      4:
        _nAx                          := _nAx + 1;
        _eState                       := E_PROGRESS.PROGRESS_BUSY;
        _fbGearInMultiMaster.Master4  := _Axes[_nMasterIndex[4]];   // assign AXIS_REF of master
    ELSE
      _eState                         := E_PROGRESS.PROGRESS_CHECK;
    END_CASE
END_CASE
CASE _eState
OF
  E_PROGRESS.PROGRESS_CHECK:
    _fbGearInMultiMaster(
                      Slave           := _AxisRef, 
                      Enable          := TRUE, 
                      GearRatio1      := _GearInParameter^[_nAxisIndex].rGearRatio[1], 
                      GearRatio2      := _GearInParameter^[_nAxisIndex].rGearRatio[2], 
                      GearRatio3      := _GearInParameter^[_nAxisIndex].rGearRatio[3], 
                      GearRatio4      := _GearInParameter^[_nAxisIndex].rGearRatio[4], 
                      Acceleration    := _GearInParameter^[_nAxisIndex].Acceleration, 
                      Deceleration    := _GearInParameter^[_nAxisIndex].Deceleration, 
                      Jerk            := _GearInParameter^[_nAxisIndex].Jerk);

    IF (_fbGearInMultiMaster.Error)
    THEN
      _nErr                           := _fbGearInMultiMaster.ErrorID;
      _stMsg.eType                    := E_MessageType.eMessageError;
      _stMsg.eDevice                  := e_Device.Axis + TO_UINT(_AxisRef.NcToPlc.AxisId);
      _stMsg.eSubdevice               := e_Subdevice.fbGearInMultiMaster;
      _stMsg.iErrorNumber             := _nErr;

      _stMsg.sText                    := concat(TO_STRING(_eCmd),'[');
      _stMsg.sText                    := concat(_stMsg.sText, TO_STRING(_nAxisIndex));
      _stMsg.sText                    := concat(_stMsg.sText, ']');
      _stMsg.sText                    := concat('fbGearInMultiMaster error: ', TO_STRING(_nErr));
      f_MessageSet(_stMsg);
      _eState                         := E_PROGRESS.PROGRESS_ERROR;

    ELSIF (_fbGearIn.InGear)
    THEN
      _eState                         := E_PROGRESS.PROGRESS_WORKING;
    END_IF

END_CASE
CASE _eState
OF
  E_PROGRESS.PROGRESS_WORKING:
    // now GearRatio[x] can be altered from outside
    // axis function waits here for further instructions from outside world
    // _stCtrl[_nAxisIndex].eProgress = e_Progress.DONE must be used to leave this axis function
    _fbGearInMultiMaster(
                      Slave           := _AxisRef, 
                      Enable          := TRUE, 
                      GearRatio1      := _GearInParameter^[_nAxisIndex].rGearRatio[1], 
                      GearRatio2      := _GearInParameter^[_nAxisIndex].rGearRatio[2], 
                      GearRatio3      := _GearInParameter^[_nAxisIndex].rGearRatio[3], 
                      GearRatio4      := _GearInParameter^[_nAxisIndex].rGearRatio[4], 
                      Acceleration    := _GearInParameter^[_nAxisIndex].Acceleration, 
                      Deceleration    := _GearInParameter^[_nAxisIndex].Deceleration, 
                      Jerk            := _GearInParameter^[_nAxisIndex].Jerk);

    IF (_fbGearInMultiMaster.Error)
    THEN
      _nErr                           := _fbGearInMultiMaster.ErrorID;
      _stMsg.eType                    := E_MessageType.eMessageError;
      _stMsg.eDevice                  := e_Device.Axis + TO_UINT(_AxisRef.NcToPlc.AxisId);
      _stMsg.eSubdevice               := e_Subdevice.fbGearInMultiMaster;
      _stMsg.iErrorNumber             := _nErr;

      _stMsg.sText                    := concat(TO_STRING(_eCmd),'[');
      _stMsg.sText                    := concat(_stMsg.sText, TO_STRING(_nAxisIndex));
      _stMsg.sText                    := concat(_stMsg.sText, ']');
      _stMsg.sText                    := concat('fbGearInMultiMaster error: ', TO_STRING(_nErr));
      f_MessageSet(_stMsg);
      _eState                         := E_PROGRESS.PROGRESS_ERROR;

    ELSIF (_Ctrl^[_nAxisIndex].eProgress = E_PROGRESS.PROGRESS_DONE)
    THEN
      // when Ctrl decides to leave; make finishing move and be done
      _eState                         := E_PROGRESS.PROGRESS_STILL_WORKING;
    END_IF
END_CASE
CASE _eState
OF
  E_PROGRESS.PROGRESS_STILL_WORKING:
    _eState                           := E_PROGRESS.PROGRESS_DONE;

    _stMsg.eType                      := E_MessageType.eMessageInfo;
    _stMsg.eDevice                    := e_Device.Axis + TO_UINT(_AxisRef.NcToPlc.AxisId);
    _stMsg.eSubdevice                 := e_Subdevice.fbGearInMultiMaster;
    _stMsg.iErrorNumber               := _eState;

    _stMsg.sText                      := concat(TO_STRING(_eCmd), ': ');
    _stMsg.sText                      := concat(_stMsg.sText, TO_STRING(_eState));
    f_MessageSet(_stMsg);
END_CASE

AxisGearInMultiMaster                 := _eState;
END_METHOD

PROPERTY AxisGearInParameter : pointer to ARRAY[1..PLC_CONSTANT.MAX_AXIS] OF ST_GEAR_IN
SET
_GearInParameter := AxisGearInParameter;
END_SET
END_PROPERTY

METHOD AxisGearOut : E_PROGRESS
VAR_INPUT
  Execute           : BOOL;
END_VAR
VAR_INST
  _eState           : E_PROGRESS;
  _rValue           : LREAL;
  _nErr             : UDINT;
  _stMsg            : ST_Message;
END_VAR
IF NOT Check() THEN AxisGearOut := E_PROGRESS.PROGRESS_ERROR; RETURN; END_IF
IF NOT Execute THEN _eState := E_PROGRESS.PROGRESS_INIT; END_IF

CASE _eState
OF
  E_PROGRESS.PROGRESS_INIT:
    IF Execute 
    THEN
      memset(ADR(_stMsg),0,SIZEOF(_stMsg));
      _nErr                       := 0;
      _rValue                     := 0;

      _fbGearOut(
            Slave                 := _AxisRef, 
            Execute               := FALSE);

      IF (_AxisRef.NcToPlc.CoupleState < 2)
      THEN
        _eState                   := E_PROGRESS.PROGRESS_DONE;
      ELSE
        _eState                   := E_PROGRESS.PROGRESS_BUSY;

        _stMsg.eType              := E_MessageType.eMessageInfo;
        _stMsg.eDevice            := e_Device.Axis + TO_UINT(_AxisRef.NcToPlc.AxisId);
        _stMsg.eSubdevice         := e_Subdevice.fbGearOut;
        _stMsg.iErrorNumber       := 0;
  
        _stMsg.sText              := concat('GearOut BUSY: ', TO_STRING(_nAxisIndex));
        f_MessageSet(_stMsg);
      END_IF
    END_IF
END_CASE
CASE _eState
OF
  E_PROGRESS.PROGRESS_BUSY:
    _fbGearOut(
            Slave                 := _AxisRef, 
            Execute               := TRUE);

    IF (_fbGearOut.Error)
    THEN
      _nErr                       := _fbGearOut.ErrorID;

      _stMsg.eType                := E_MessageType.eMessageError;
      _stMsg.eDevice              := e_Device.Axis + TO_UINT(_AxisRef.NcToPlc.AxisId);
      _stMsg.eSubdevice           := e_Subdevice.fbGearOut;
      _stMsg.iErrorNumber         := _nErr;

      _stMsg.sText                := concat('GearOut ERROR: ', TO_STRING(_nAxisIndex));
      f_MessageSet(_stMsg);
      _eState                     := E_PROGRESS.PROGRESS_ERROR;

    ELSIF (_fbGearOut.Done)
    THEN
      _stMsg.eType                := E_MessageType.eMessageInfo;
      _stMsg.eDevice              := e_Device.Axis + TO_UINT(_AxisRef.NcToPlc.AxisId);
      _stMsg.eSubdevice           := e_Subdevice.fbGearOut;
      _stMsg.iErrorNumber         := 0;
  
      _stMsg.sText                := concat('GearOut DONE: ', TO_STRING(_nAxisIndex));
      f_MessageSet(_stMsg);

      IF (_AxisRef.NcToPlc.CoupleState < 2)
      THEN
        _eState                   := E_PROGRESS.PROGRESS_DONE;
      ELSE
        _eState                   := E_PROGRESS.PROGRESS_STARTUP;
      END_IF
    END_IF
END_CASE
CASE _eState
OF
  E_PROGRESS.PROGRESS_STARTUP:
    _eState                       := E_PROGRESS.PROGRESS_BUSY;
    _fbGearOut(
          Slave                   := _AxisRef, 
          Execute                 := FALSE);

    _stMsg.eType                  := E_MessageType.eMessageInfo;
    _stMsg.eDevice                := e_Device.Axis + TO_UINT(_AxisRef.NcToPlc.AxisId);
    _stMsg.eSubdevice             := e_Subdevice.fbGearOut;
    _stMsg.iErrorNumber           := 0;

    _stMsg.sText                  := concat('GearOut CoupleState: ', TO_STRING(_AxisRef.NcToPlc.CoupleState));
    f_MessageSet(_stMsg);
END_CASE
CASE _eState
OF
  E_PROGRESS.PROGRESS_DONE,
  E_PROGRESS.PROGRESS_ERROR:
    _fbGearOut(
            Slave                 := _AxisRef, 
            Execute               := FALSE);
END_CASE

AxisGearOut                       := _eState;
END_METHOD

METHOD AxisHalt : E_PROGRESS
VAR_INPUT
  Execute           : BOOL;
  Data              : ST_AXIS_MOVE_DATA;
END_VAR
VAR_INST
  _eres,
  _eState           : E_PROGRESS;
  _rValue           : LREAL;
  _udiErr           : UDINT;
  _stMsg            : ST_Message;


END_VAR
IF NOT Check() THEN AxisHalt := E_PROGRESS.PROGRESS_ERROR; RETURN; END_IF
IF NOT Execute THEN _eState := E_PROGRESS.PROGRESS_INIT; END_IF

CASE _eState
OF
  E_PROGRESS.PROGRESS_INIT:
    IF Execute 
    THEN
      memset(ADR(_stMsg),0,SIZEOF(_stMsg));
      _udiErr       := 0;
      _rValue       := 0;
      _eState       := E_PROGRESS.PROGRESS_BUSY;
    END_IF
END_CASE
CASE _eState
OF
  E_PROGRESS.PROGRESS_BUSY:
    _eState         := E_PROGRESS.PROGRESS_OCCUPIED;
    _eres           := Halt(
                            Execute := FALSE, 
                            Dec     := Data.rDec, 
                            Jerk    := Data.rJerk);
END_CASE
CASE _eState
OF
  E_PROGRESS.PROGRESS_OCCUPIED:
    _eres           := Halt(
                            Execute := TRUE, 
                            Dec     := Data.rDec, 
                            Jerk    := Data.rJerk);

    IF (_eres = E_PROGRESS.PROGRESS_ERROR)
    THEN
        _eState     := E_PROGRESS.PROGRESS_ERROR;
    ELSIF (_eres = E_PROGRESS.PROGRESS_DONE)
    THEN 
      _eState       := E_PROGRESS.PROGRESS_WORKING;
    END_IF
END_CASE
CASE _eState
OF
  E_PROGRESS.PROGRESS_WORKING:
    _eState         := E_PROGRESS.PROGRESS_DONE;
    _eres           := Halt(
                            Execute := FALSE, 
                            Dec     := Data.rDec, 
                            Jerk    := Data.rJerk);
END_CASE

AxisHalt := _eState;
END_METHOD

METHOD AxisHome : E_PROGRESS
VAR_INPUT
  Execute           : BOOL;
END_VAR
VAR_INST
  _eres,
  _eState           : E_PROGRESS;
  _rValue           : LREAL;
  _udiErr           : UDINT;
  _stMsg            : ST_Message;


END_VAR
IF NOT Check() THEN AxisHome := E_PROGRESS.PROGRESS_ERROR; RETURN; END_IF
IF NOT Execute THEN _eState := E_PROGRESS.PROGRESS_INIT; END_IF

CASE _eState
OF
  E_PROGRESS.PROGRESS_INIT:
    IF Execute 
    THEN
      memset(ADR(_stMsg),0,SIZEOF(_stMsg));
      _udiErr               := 0;
      _rValue               := 0;

      IF (_AxisRef.Status.Homed)
      THEN
        _eState             := E_PROGRESS.PROGRESS_BUSY;
      ELSE
        _eState             := E_PROGRESS.PROGRESS_PREPARE;
      END_IF
    END_IF
END_CASE
CASE _eState
OF
  E_PROGRESS.PROGRESS_BUSY:
    _eState                 := E_PROGRESS.PROGRESS_STARTUP;
    _eres                   := Home(
                                    Execute   := FALSE,
                                    Position  := _HomeParameter^[_nAxisIndex].stHomingParam.Position,
                                    HomingMode:= Tc2_MC2.MC_HomingMode.MC_ResetCalibration,
                                    Options   := _HomeParameter^[_nAxisIndex].stHomingParam.Options);
END_CASE
CASE _eState
OF
  E_PROGRESS.PROGRESS_STARTUP:
    _Info^[_nAxisIndex].bReferenced   := FALSE;

    _eres                   := Home(
                                    Execute   := TRUE,
                                    Position  := _HomeParameter^[_nAxisIndex].stHomingParam.Position,
                                    HomingMode:= Tc2_MC2.MC_HomingMode.MC_ResetCalibration,
                                    Options   := _HomeParameter^[_nAxisIndex].stHomingParam.Options);
    IF (_eres = E_PROGRESS.PROGRESS_DONE)
    THEN
      _eState               := E_PROGRESS.PROGRESS_PREPARE;
    END_IF
END_CASE
CASE _eState
OF
  E_PROGRESS.PROGRESS_PREPARE:
      _eState               := E_PROGRESS.PROGRESS_CHECK;

      _eres                 := Home(
                                    Execute   := FALSE,
                                    Position  := _HomeParameter^[_nAxisIndex].stHomingParam.Position,
                                    HomingMode:= Tc2_MC2.MC_HomingMode.MC_ResetCalibration,
                                    Options   := _HomeParameter^[_nAxisIndex].stHomingParam.Options);
END_CASE
CASE _eState
OF
  E_PROGRESS.PROGRESS_CHECK:
    _eState                 := E_PROGRESS.PROGRESS_OCCUPIED;

END_CASE
CASE _eState
OF
  E_PROGRESS.PROGRESS_OCCUPIED:
    _eres                   := Home(
                                    Execute   := TRUE,
                                    Position  := _HomeParameter^[_nAxisIndex].stHomingParam.Position,
                                    HomingMode:= _HomeParameter^[_nAxisIndex].stHomingParam.HomingMode,
                                    Options   := _HomeParameter^[_nAxisIndex].stHomingParam.Options);

    IF (_eres = E_PROGRESS.PROGRESS_ERROR)
    THEN
      _eState               := E_PROGRESS.PROGRESS_ERROR;
    ELSIF (_eres = E_PROGRESS.PROGRESS_DONE)
    THEN
      _eState               := E_PROGRESS.PROGRESS_WORKING;
    END_IF
END_CASE
CASE _eState
OF
  E_PROGRESS.PROGRESS_WORKING:
    _eState                 := E_PROGRESS.PROGRESS_DONE;

    _eres                   := Home(
                                    Execute   := FALSE,
                                    Position  := _HomeParameter^[_nAxisIndex].stHomingParam.Position,
                                    HomingMode:= _HomeParameter^[_nAxisIndex].stHomingParam.HomingMode,
                                    Options   := _HomeParameter^[_nAxisIndex].stHomingParam.Options);
END_CASE

AxisHome := _eState;
END_METHOD

METHOD AxisIdle : E_PROGRESS
VAR_INPUT
  Execute           : BOOL;
END_VAR
VAR_INST
  _eResult,
  _eState           : E_PROGRESS;
  _stMsg            : ST_Message;
  _nRetry           : UINT;
END_VAR
IF NOT Check() THEN AxisIdle := E_PROGRESS.PROGRESS_ERROR; return; END_IF
IF NOT Execute THEN _eState := E_PROGRESS.PROGRESS_INIT; END_IF

CASE _eState
OF
  E_PROGRESS.PROGRESS_INIT:
    IF Execute 
    THEN
      memset(ADR(_stMsg),0,SIZEOF(_stMsg));
      _nRetry                       := 0;
      _eResult                      := Reset(FALSE);
      _eState                       := E_PROGRESS.PROGRESS_BUSY;
    END_IF
END_CASE
CASE _eState
OF
  E_PROGRESS.PROGRESS_BUSY:
    _eResult                        := Reset(TRUE);

    IF (_eResult = E_PROGRESS.PROGRESS_DONE)
    THEN
      _nRetry                       := _nRetry + 1;
      _eState                       := E_PROGRESS.PROGRESS_STARTUP;
    END_IF
END_CASE
CASE _eState
OF
  E_PROGRESS.PROGRESS_STARTUP:
    _eResult                        := Reset(FALSE);
    _eResult                        := Enable(FALSE);
    _eState                         := E_PROGRESS.PROGRESS_CHECK;
END_CASE
CASE _eState
OF
  E_PROGRESS.PROGRESS_PREPARE:
    _eResult                        := Reset(FALSE);
    _eResult                        := Enable(FALSE);

    _eState                         := E_PROGRESS.PROGRESS_BUSY;

    _stMsg.eType                    := E_MessageType.eMessageInfo;
    _stMsg.eDevice                  := e_Device.Axis + (_AxisRef.NcToPlc.AxisId);
    _stMsg.eSubdevice               :=  e_SubDevice.AxisIdle;
    _stMsg.iErrorNumber             := _nErrorId;

    _stMsg.sText                    := concat(TO_STRING(_eCmd), ' retry: ');
    _stMsg.sText                    := concat(_stMsg.sText, TO_STRING(_nRetry));

    f_MessageSet(_stMsg);
END_CASE
CASE _eState
OF
  E_PROGRESS.PROGRESS_CHECK:
    _eResult                        := Enable(TRUE);

    IF (_nRetry > MAX_RETRY)
    THEN
      _eState                       := E_PROGRESS.PROGRESS_ERROR;

    ELSIF (_eResult = E_PROGRESS.PROGRESS_DONE)
    THEN
      Enable(FALSE);
      _eState                       := E_PROGRESS.PROGRESS_DONE;

    ELSIF (_eResult = E_PROGRESS.PROGRESS_ERROR)
    THEN
      _eState                       := E_PROGRESS.PROGRESS_PREPARE;

      _nErrorId                     := _AxisRef.NcToPlc.ErrorCode;
    
      _stMsg.eType                  := E_MessageType.eMessageError;
      _stMsg.eDevice                := e_Device.Axis + (_AxisRef.NcToPlc.AxisId);
      _stMsg.eSubdevice             :=  e_SubDevice.AxisIdle;
      _stMsg.iErrorNumber           := _nErrorId;

      _stMsg.sText                  := concat(TO_STRING(_eCmd), ' error axis enable: ');
      _stMsg.sText                  := concat(_stMsg.sText, TO_STRING(_nAxisIndex));

      f_MessageSet(_stMsg);
    END_IF
END_CASE

AxisIdle                                := _eState;
END_METHOD

PROPERTY AxisIndex : uint
SET
_nAxisIndex := AxisIndex;
END_SET
END_PROPERTY

PROPERTY AxisInfo : pointer to ARRAY[1..PLC_CONSTANT.MAX_AXIS] OF ST_AXIS_INFO
SET
_Info := AxisInfo;
END_SET
END_PROPERTY

METHOD PRIVATE AxisInit : E_PROGRESS
VAR_INPUT
  Execute           : BOOL;
END_VAR
VAR_INST
  _eResult,
  _eState           : E_PROGRESS;
  _rValue           : LREAL;
  _stMsg            : ST_Message;
END_VAR
IF NOT Check() THEN AxisInit := E_PROGRESS.PROGRESS_ERROR; RETURN; END_IF
IF NOT Execute THEN _eState := E_PROGRESS.PROGRESS_INIT; END_IF

CASE _eState
OF
  E_PROGRESS.PROGRESS_INIT:
    IF Execute 
    THEN
      memset(ADR(_stMsg),0,SIZEOF(_stMsg));

      _nErrorId                     := 0;
      _rValue                       := 0;
      _eState                       := E_PROGRESS.PROGRESS_BUSY;
      _eInit                        := _eState;
    END_IF
END_CASE
CASE _eState
OF
  E_PROGRESS.PROGRESS_BUSY:
    _eState                         := E_PROGRESS.PROGRESS_STARTUP;
    _eResult                        := StartUp(FALSE);
END_CASE
CASE _eState
OF
  E_PROGRESS.PROGRESS_STARTUP:
    _eResult                        := StartUp(TRUE);
    IF (_eResult = E_PROGRESS.PROGRESS_DONE)
    THEN
      _eState                       := E_PROGRESS.PROGRESS_PREPARE;
      _eResult                      := AxisReset(FALSE);
    ELSIF (_eResult = E_PROGRESS.PROGRESS_ERROR)
    THEN
      _eState                       := _eResult;

      _stMsg.eType                  := E_MessageType.eMessageError;
      _stMsg.eDevice                := e_Device.Axis + (_AxisRef.NcToPlc.AxisId);
      _stMsg.eSubdevice             := e_Subdevice.AxisStartUp;
      _stMsg.iErrorNumber := _nErrorId  := 6666;

      _stMsg.sText                  := TO_STRING(_eState);
      f_MessageSet(_stMsg);

    END_IF
END_CASE
CASE _eState
OF
  E_PROGRESS.PROGRESS_PREPARE:
    _eResult                        := AxisReset(TRUE);
    IF (_eResult = E_PROGRESS.PROGRESS_DONE)
    THEN
      _fbCoeRead(
                Execute             := FALSE,
                NetId               := _AxisRef.ADS.NetId, 
                Axis                := _AxisRef);
  
      IF (EncoderType > 1)
      THEN
        memset(ADR(_sDeviceName),0,SIZEOF(_sDeviceName));
  
        _eState                     := E_PROGRESS.PROGRESS_CHECK;
      ELSE
        _sDeviceName                := _sAxisName;
        _eState                     := E_PROGRESS.PROGRESS_WORKING;
      END_IF
    ELSIF (_eResult = E_PROGRESS.PROGRESS_ERROR)
    THEN
      _eState                       := _eResult;

      _stMsg.eType                  := E_MessageType.eMessageError;
      _stMsg.eDevice                := e_Device.Axis + (_AxisRef.NcToPlc.AxisId);
      _stMsg.eSubdevice             := e_Subdevice.AxisStartUp;
      _stMsg.iErrorNumber           := ErrorId;

      _stMsg.sText                  := TO_STRING(_eState);
      f_MessageSet(_stMsg);

    END_IF
END_CASE
CASE _eState
OF
  E_PROGRESS.PROGRESS_CHECK:
    _eResult                        := AxisReset(FALSE);
    // get manufacturer device name in CoE
    _fbCoeRead.Index                := 16#1008;
    _fbCoeRead.SubIndex             := 0;
    _fbCoeRead.pDstBuf              := ADR(_sDeviceName);
    _fbCoeRead.BufLen               := SIZEOF(_sDeviceName);

    _fbCoeRead(
              Execute               := TRUE,
              NetId                 := _AxisRef.ADS.NetId, 
              Axis                  := _AxisRef);

    IF _fbCoeRead.Busy
    THEN
      _eState                       := E_PROGRESS.PROGRESS_OCCUPIED;
    END_IF
END_CASE
CASE _eState
OF
  E_PROGRESS.PROGRESS_OCCUPIED:
    _fbCoeRead(
              NetId                 := _AxisRef.ADS.NetId, 
              Axis                  := _AxisRef);

    IF NOT _fbCoeRead.Busy
    THEN
      _eState                       := E_PROGRESS.PROGRESS_WORKING;
    END_IF

// in case encoder type is used without hardware, error must be ignored here
(*
    IF (_fbCoeRead.Error)
    THEN
      _eState                       := E_PROGRESS.ERROR;

      _Info^[_nAxisIndex].nErrorId  := SEL((_fbCoeRead.CANopenErrId > 0), _fbCoeRead.AdsErrId, _fbCoeRead.CANopenErrId);

      _stMsg.eType                  := E_MessageType.eMessageError;
      _stMsg.eDevice                := e_Device.Axis + TO_DINT(_AxisRef.NcToPlc.AxisId);
      _stMsg.eSubdevice             := e_Subdevice.fbCoeRead;

      _stMsg.iErrorNumber           := SEL((_fbCoeRead.CANopenErrId > 0), _fbCoeRead.AdsErrId, _fbCoeRead.CANopenErrId);

      _stMsg.sText                  := TO_STRING(_eState);
      f_MessageSet(_stMsg);

      _fbCoeRead(
                Execute             := FALSE,
                NetId               := _AxisRef.ADS.NetId, 
                Axis                := _AxisRef);

    ELSIF NOT _fbCoeRead.Busy
    THEN
      _eState                       := E_PROGRESS.WORKING;
    END_IF
*)
END_CASE
CASE _eState
OF
  E_PROGRESS.PROGRESS_WORKING:
    _eState                         := E_PROGRESS.PROGRESS_DONE;
    // set default for axis release
    AxisEnableNegative              := TRUE;
    AxisEnablePositive              := TRUE;

    // clear fb
    _fbCoeRead(
              Execute               := FALSE,
              NetId                 := _AxisRef.ADS.NetId, 
              Axis                  := _AxisRef);

    _stMsg.eType                    := E_MessageType.eMessageInfo;
    _stMsg.eDevice                  := e_Device.Axis + (_AxisRef.NcToPlc.AxisId);
    _stMsg.eSubdevice               := e_Subdevice.AxisStartUp;
    _stMsg.iErrorNumber             := 0;
    _stMsg.sText                    := concat('Axis Init: ', _sDeviceName);
    _stMsg.sText                    := concat(_stMsg.sText, ' : ');
    _stMsg.sText                    := concat(_stMsg.sText, TO_STRING(_eState));

  IF (_MessageLevel > E_MessageType.eMessageError)
  THEN
    f_MessageSet(_stMsg);
  END_IF
END_CASE

AxisInit                            := _eState;
END_METHOD

METHOD AxisMoveToPosition : E_PROGRESS
VAR_INPUT
  Execute           : BOOL;
  Data              : ST_AXIS_MOVE_DATA;
END_VAR
VAR_INST
  _eres,
  _eState           : E_PROGRESS;
END_VAR
IF NOT Check() THEN AxisMoveToPosition := E_PROGRESS.PROGRESS_ERROR; RETURN; END_IF
IF NOT Execute THEN _eState := E_PROGRESS.PROGRESS_INIT; END_IF

CASE _eState
OF
  E_PROGRESS.PROGRESS_INIT:
    IF Execute 
    THEN
      _eState               := E_PROGRESS.PROGRESS_BUSY;
    END_IF
END_CASE
CASE _eState
OF
  E_PROGRESS.PROGRESS_BUSY:
    _eState                 := E_PROGRESS.PROGRESS_OCCUPIED;
    _eres                   := MoveToPos(
                                      Execute    := FALSE, 
                                      Position   := Data.rSetPos, 
                                      Vel        := Data.rSetVelo, 
                                      Acc        := Data.rAcc, 
                                      Dec        := Data.rDec, 
                                      Jerk       := Data.rJerk, 
                                      BufferMode := Tc2_MC2.MC_BufferMode.MC_Aborting);
END_CASE
CASE _eState
OF
  E_PROGRESS.PROGRESS_OCCUPIED:
    _eres                   := MoveToPos(
                                      Execute    := TRUE, 
                                      Position   := Data.rSetPos, 
                                      Vel        := Data.rSetVelo, 
                                      Acc        := Data.rAcc, 
                                      Dec        := Data.rDec, 
                                      Jerk       := Data.rJerk, 
                                      BufferMode := Tc2_MC2.MC_BufferMode.MC_Aborting);

    IF (_eres = E_PROGRESS.PROGRESS_ERROR)
    THEN
        _eState             := E_PROGRESS.PROGRESS_ERROR;
    ELSIF (_eres = E_PROGRESS.PROGRESS_DONE)
    THEN 
      _eState               := E_PROGRESS.PROGRESS_WORKING;
    END_IF
END_CASE
CASE _eState
OF
  E_PROGRESS.PROGRESS_WORKING:
    _eState                 := E_PROGRESS.PROGRESS_DONE;
    _eres                   := MoveToPos(
                                      Execute    := FALSE, 
                                      Position   := Data.rSetPos, 
                                      Vel        := Data.rSetVelo, 
                                      Acc        := Data.rAcc, 
                                      Dec        := Data.rDec, 
                                      Jerk       := Data.rJerk, 
                                      BufferMode := Tc2_MC2.MC_BufferMode.MC_Aborting);
END_CASE

AxisMoveToPosition := _eState;
END_METHOD

METHOD AxisMoveVelocity : E_PROGRESS
VAR_INPUT
  Execute           : BOOL;
  Data              : ST_AXIS_MOVE_DATA;
END_VAR
VAR_INST
  _eres,
  _eState           : E_PROGRESS;
END_VAR
IF NOT Check() THEN AxisMoveVelocity := E_PROGRESS.PROGRESS_ERROR; RETURN; END_IF
IF NOT Execute THEN _eState := E_PROGRESS.PROGRESS_INIT; END_IF

CASE _eState
OF
  E_PROGRESS.PROGRESS_INIT:
    IF Execute 
    THEN
      _eState               := E_PROGRESS.PROGRESS_BUSY;
    END_IF
END_CASE
CASE _eState
OF
  E_PROGRESS.PROGRESS_BUSY:
    _eState                 := E_PROGRESS.PROGRESS_OCCUPIED;
    _eres                   := MoveVelo(
                                    Execute     := FALSE, 
                                    Velocity    := Data.rSetVelo, 
                                    Acc         := Data.rAcc, 
                                    Dec         := Data.rDec, 
                                    Jerk        := Data.rJerk, 
                                    Direction   := Data.iDirection, 
                                    BufferMode  := Tc2_MC2.MC_BufferMode.MC_Aborting);
END_CASE
CASE _eState
OF
  E_PROGRESS.PROGRESS_OCCUPIED:
    _eres                   := MoveVelo(
                                    Execute     := TRUE, 
                                    Velocity    := Data.rSetVelo, 
                                    Acc         := Data.rAcc, 
                                    Dec         := Data.rDec, 
                                    Jerk        := Data.rJerk, 
                                    Direction   := Data.iDirection, 
                                    BufferMode  := Tc2_MC2.MC_BufferMode.MC_Aborting);
    IF (_eres = E_PROGRESS.PROGRESS_ERROR)
    THEN
        _eState             := E_PROGRESS.PROGRESS_ERROR;
    ELSIF (_eres = E_PROGRESS.PROGRESS_DONE)
    THEN 
      _eState               := E_PROGRESS.PROGRESS_WORKING;
    END_IF
END_CASE
CASE _eState
OF
  E_PROGRESS.PROGRESS_WORKING:
    _eState                 := E_PROGRESS.PROGRESS_DONE;
    _eres                   := MoveVelo(
                                    Execute     := FALSE, 
                                    Velocity    := Data.rSetVelo, 
                                    Acc         := Data.rAcc, 
                                    Dec         := Data.rDec, 
                                    Jerk        := Data.rJerk, 
                                    Direction   := Data.iDirection, 
                                    BufferMode  := Tc2_MC2.MC_BufferMode.MC_Aborting);
END_CASE

AxisMoveVelocity                := _eState;
END_METHOD

METHOD AxisParameterRead : E_PROGRESS
VAR_INPUT
  Execute           : BOOL;
  ParameterNr       : Tc2_MC2.MC_AxisParameter;
END_VAR
VAR_INST
  _eres,
  _eState           : E_PROGRESS;
  _rValue           : LREAL;
  _eParam           : Tc2_MC2.MC_AxisParameter;
END_VAR
IF NOT Check() THEN AxisParameterRead := E_PROGRESS.PROGRESS_ERROR; RETURN; END_IF
IF NOT Execute THEN _eState := E_PROGRESS.PROGRESS_INIT; END_IF

CASE _eState
OF
  E_PROGRESS.PROGRESS_INIT:
    IF Execute 
    THEN
      _rValue                                     := 0.0;
      _eParam                                     := ParameterNr;
      _eState                                     := E_PROGRESS.PROGRESS_BUSY;
    END_IF
END_CASE
CASE _eState
OF
  E_PROGRESS.PROGRESS_BUSY:
    _eState                                       := E_PROGRESS.PROGRESS_OCCUPIED;
    _eres           := ReadParameter(
                                  Execute         := FALSE,
                                  ParameterNumber := _eParam);
END_CASE
CASE _eState
OF
  E_PROGRESS.PROGRESS_OCCUPIED:
    _eres           := ReadParameter(
                                  Execute         := TRUE,
                                  ParameterNumber := _eParam);

    IF (_eres = E_PROGRESS.PROGRESS_ERROR)
    THEN
      _eState                                     := E_PROGRESS.PROGRESS_ERROR;
    ELSIF (_eres = E_PROGRESS.PROGRESS_DONE)
    THEN 
      _eState                                     := E_PROGRESS.PROGRESS_WORKING;
    END_IF

  E_PROGRESS.PROGRESS_WORKING:
    _eState                                       := E_PROGRESS.PROGRESS_DONE;
    _eres           := ReadParameter(
                                  Execute         := FALSE,
                                  ParameterNumber := _eParam);

    _eParameterNrRead                             :=
    _NcParameterOut^[_nAxisIndex].ParameterNumber := _eParam;

    _NcParameterOut^[_nAxisIndex].rValue          :=
    _rParameterReadValue                          := 
    _rValue                                       := _rValueParameterRead;
END_CASE

AxisParameterRead := _eState;
END_METHOD

METHOD AxisParameterWrite : E_PROGRESS
VAR_INPUT
  Execute           : BOOL;
  ParameterNr       : Tc2_MC2.MC_AxisParameter;
END_VAR
VAR_INST
  _eres,
  _eState           : E_PROGRESS;
  _rValue           : LREAL;
  _eParam           : Tc2_MC2.MC_AxisParameter;
END_VAR
IF NOT Check() THEN AxisParameterWrite := E_PROGRESS.PROGRESS_ERROR; RETURN; END_IF
IF NOT Execute THEN _eState := E_PROGRESS.PROGRESS_INIT; END_IF

CASE _eState
OF
  E_PROGRESS.PROGRESS_INIT:
    IF Execute 
    THEN
      _rValue                                     := _rParameterWrtValue;
      _eParam                                     := ParameterNr;
      _eState                                     := E_PROGRESS.PROGRESS_BUSY;
    END_IF
END_CASE
CASE _eState
OF
  E_PROGRESS.PROGRESS_BUSY:
    _eState                                       := E_PROGRESS.PROGRESS_OCCUPIED;
    _eres           := WriteParameter(
                                  Execute         := FALSE,
                                  Value           := _rValue,
                                  ParameterNumber := _eParam);
END_CASE
CASE _eState
OF
  E_PROGRESS.PROGRESS_OCCUPIED:
    _eres           := WriteParameter(
                                  Execute         := TRUE,
                                  Value           := _rValue,
                                  ParameterNumber := _eParam);
    IF (_eres = E_PROGRESS.PROGRESS_ERROR)
    THEN
      _eState                                     := E_PROGRESS.PROGRESS_ERROR;
    ELSIF (_eres = E_PROGRESS.PROGRESS_DONE)
    THEN
      _NcParameterOut^[_nAxisIndex].rValue          := _rValue;
      _NcParameterOut^[_nAxisIndex].ParameterNumber := _eParam;
      _eState                                       := E_PROGRESS.PROGRESS_WORKING;
    END_IF

  E_PROGRESS.PROGRESS_WORKING:
    _eState                                       := E_PROGRESS.PROGRESS_DONE;
    _eres           := WriteParameter(
                                  Execute         := FALSE,
                                  Value           := _rValue,
                                  ParameterNumber := _eParam);
END_CASE

AxisParameterWrite                                    := _eState;
END_METHOD

METHOD AxisParameterWritePersistent : E_PROGRESS
VAR_INPUT
  Execute           : BOOL;
  ParameterNr       : Tc2_MC2.MC_AxisParameter;
END_VAR
VAR_INST
  _eres,
  _eState           : E_PROGRESS;
  _rValue           : LREAL;
END_VAR
IF NOT Check() THEN AxisParameterWritePersistent := E_PROGRESS.PROGRESS_ERROR; RETURN; END_IF
IF NOT Execute THEN _eState := E_PROGRESS.PROGRESS_INIT; END_IF

CASE _eState
OF
  E_PROGRESS.PROGRESS_INIT:
    IF Execute 
    THEN
      _rValue                                     := _rParameterWrtValue;
      _eState                                     := E_PROGRESS.PROGRESS_BUSY;
    END_IF
END_CASE
CASE _eState
OF
  E_PROGRESS.PROGRESS_BUSY:
    _eState                                       := E_PROGRESS.PROGRESS_OCCUPIED;
    _eres           := WriteParameterPersistent(
                                  Execute         := FALSE,
                                  Value           := _rValue,
                                  ParameterNumber := ParameterNr);
END_CASE
CASE _eState
OF
  E_PROGRESS.PROGRESS_OCCUPIED:
    _eres           := WriteParameterPersistent(
                                  Execute         := TRUE,
                                  Value           := _rValue,
                                  ParameterNumber := ParameterNr);
    IF (_eres = E_PROGRESS.PROGRESS_ERROR)
    THEN
      _eState                                     := E_PROGRESS.PROGRESS_ERROR;
    ELSIF (_eres = E_PROGRESS.PROGRESS_DONE)
    THEN 
      _eState                                     := E_PROGRESS.PROGRESS_WORKING;
    END_IF

  E_PROGRESS.PROGRESS_WORKING:
    _eState                                       := E_PROGRESS.PROGRESS_DONE;
    _eres           := WriteParameterPersistent(
                                  Execute         := FALSE,
                                  Value           := _rValue,
                                  ParameterNumber := ParameterNr);
END_CASE

AxisParameterWritePersistent                          := _eState;
END_METHOD

METHOD AxisReset : E_PROGRESS
VAR_INPUT
  Execute           : BOOL;
END_VAR
VAR_INST
  _eres,
  _eState           : E_PROGRESS;
END_VAR
IF NOT Check() THEN AxisReset := E_PROGRESS.PROGRESS_ERROR; RETURN; END_IF
IF NOT Execute THEN _eState := E_PROGRESS.PROGRESS_INIT; END_IF

CASE _eState
OF
  E_PROGRESS.PROGRESS_INIT:
    IF Execute 
    THEN
      _eState                       := E_PROGRESS.PROGRESS_BUSY;
    END_IF
END_CASE
CASE _eState
OF
  E_PROGRESS.PROGRESS_BUSY:
    _eres                           := Reset(FALSE);
    _eState                         := E_PROGRESS.PROGRESS_OCCUPIED;
END_CASE
CASE _eState
OF
  E_PROGRESS.PROGRESS_OCCUPIED:
    _eres                           := Reset(TRUE);
    IF (_eres = E_PROGRESS.PROGRESS_DONE)
    THEN
      _eState                       := E_PROGRESS.PROGRESS_WORKING;
    ELSIF (_eres = E_PROGRESS.PROGRESS_ERROR)
    THEN
      _eState                       := E_PROGRESS.PROGRESS_ERROR;
    END_IF
END_CASE
CASE _eState
OF
  E_PROGRESS.PROGRESS_WORKING:
    _eres                           := Reset(FALSE);
    _eState                         := E_PROGRESS.PROGRESS_DONE;
END_CASE

AxisReset                           := _eState;
END_METHOD

METHOD AxisSendToPosition : E_PROGRESS
VAR_INPUT
  Execute           : BOOL;
  Data              : ST_AXIS_MOVE_DATA;
END_VAR
VAR_INST
  _eres,
  _eState           : E_PROGRESS;
END_VAR
IF NOT Check() THEN AxisSendToPosition := E_PROGRESS.PROGRESS_ERROR; RETURN; END_IF
IF NOT Execute THEN _eState := E_PROGRESS.PROGRESS_INIT; END_IF

CASE _eState
OF
  E_PROGRESS.PROGRESS_INIT:
    IF Execute 
    THEN
      _eState               := E_PROGRESS.PROGRESS_BUSY;
    END_IF
END_CASE
CASE _eState
OF
  E_PROGRESS.PROGRESS_BUSY:
    _eState                 := E_PROGRESS.PROGRESS_OCCUPIED;
    _eres                   := SendToPos(
                                      Execute    := FALSE, 
                                      Position   := Data.rSetPos, 
	                                    Distance   := _MotionOptions^[_nAxisIndex].rDistance, 
                                      Vel        := Data.rSetVelo, 
                                      Acc        := Data.rAcc, 
                                      Dec        := Data.rDec, 
                                      Jerk       := Data.rJerk, 
	                                    BufferMode := Tc2_MC2.MC_BufferMode.MC_Aborting);
END_CASE
CASE _eState
OF
  E_PROGRESS.PROGRESS_OCCUPIED:
    _eres                   := SendToPos(
                                      Execute    := TRUE, 
                                      Position   := Data.rSetPos, 
	                                    Distance   := _MotionOptions^[_nAxisIndex].rDistance, 
                                      Vel        := Data.rSetVelo, 
                                      Acc        := Data.rAcc, 
                                      Dec        := Data.rDec, 
                                      Jerk       := Data.rJerk, 
	                                    BufferMode := Tc2_MC2.MC_BufferMode.MC_Aborting);

    IF (_eres = E_PROGRESS.PROGRESS_ERROR)
    THEN
        _eState             := E_PROGRESS.PROGRESS_ERROR;
    ELSIF (_eres = E_PROGRESS.PROGRESS_DONE)
    THEN 
      _eState               := E_PROGRESS.PROGRESS_WORKING;
    END_IF
END_CASE
CASE _eState
OF
  E_PROGRESS.PROGRESS_WORKING:
    _eState                 := E_PROGRESS.PROGRESS_DONE;
    _eres                   := SendToPos(
                                      Execute    := FALSE, 
                                      Position   := Data.rSetPos, 
	                                    Distance   := _MotionOptions^[_nAxisIndex].rDistance, 
                                      Vel        := Data.rSetVelo, 
                                      Acc        := Data.rAcc, 
                                      Dec        := Data.rDec, 
                                      Jerk       := Data.rJerk, 
	                                    BufferMode := Tc2_MC2.MC_BufferMode.MC_Aborting);
END_CASE

AxisSendToPosition := _eState;
END_METHOD

PROPERTY AxisState : pointer to ARRAY[1..PLC_CONSTANT.MAX_AXIS] OF ST_AXIS_STATE
SET
_State := AxisState;
END_SET
END_PROPERTY

METHOD AxisStop : E_PROGRESS
VAR_INPUT
  Execute           : BOOL;
  Data              : ST_AXIS_MOVE_DATA;
END_VAR
VAR_INST
  _eres,
  _eState           : E_PROGRESS;
END_VAR
IF NOT Check() THEN AxisStop := E_PROGRESS.PROGRESS_ERROR; RETURN; END_IF
IF NOT Execute THEN _eState := E_PROGRESS.PROGRESS_INIT; END_IF

CASE _eState
OF
  E_PROGRESS.PROGRESS_INIT:
    IF Execute 
    THEN
      _eState       := E_PROGRESS.PROGRESS_BUSY;
    END_IF
END_CASE
CASE _eState
OF
  E_PROGRESS.PROGRESS_BUSY:
    _eState         := E_PROGRESS.PROGRESS_OCCUPIED;
    _eres           := Stop(
                            Execute := FALSE, 
                            Dec     := Data.rDec, 
                            Jerk    := Data.rJerk);
END_CASE
CASE _eState
OF
  E_PROGRESS.PROGRESS_OCCUPIED:
    _eres           := Stop(
                            Execute := TRUE, 
                            Dec     := Data.rDec, 
                            Jerk    := Data.rJerk);

    IF (_eres = E_PROGRESS.PROGRESS_ERROR)
    THEN
        _eState     := E_PROGRESS.PROGRESS_ERROR;
    ELSIF (_eres = E_PROGRESS.PROGRESS_DONE)
    THEN 
      _eState       := E_PROGRESS.PROGRESS_WORKING;
    END_IF
END_CASE
CASE _eState
OF
  E_PROGRESS.PROGRESS_WORKING:
    _eState         := E_PROGRESS.PROGRESS_DONE;
    _eres           := Stop(
                            Execute := FALSE, 
                            Dec     := Data.rDec, 
                            Jerk    := Data.rJerk);
END_CASE

AxisStop := _eState;
END_METHOD

METHOD PRIVATE Check : BOOL
//-----------------------------------------------------------------------------
IF (_nAxisIndex < 1) OR
   (_nAxisIndex > PLC_CONSTANT.MAX_AXIS)
THEN
  _eCheck                 := E_CHECK_STATE.AXIS_INDEX_OUT_OF_RANGE;
  RETURN;
END_IF

IF NOT __ISVALIDREF(_Axes)
THEN
  _eCheck                 := E_CHECK_STATE.AXIS_REF_POINTER_INVALID;
  RETURN;
END_IF
//-----------------------------------------------------------------------------
// get my AXIS_REF pointer for use in base class
//-----------------------------------------------------------------------------
_AxisRef                  REF= _Axes[_nAxisIndex];
//-----------------------------------------------------------------------------

IF NOT (_Ctrl <> 0)
THEN
  _eCheck                 := E_CHECK_STATE.AXIS_CTRL_POINTER_INVALID;
  RETURN;
END_IF

IF NOT (_State <> 0)
THEN
  _eCheck                 := E_CHECK_STATE.AXIS_STATE_POINTER_INVALID;
  RETURN;
END_IF

IF NOT (_Info <> 0)
THEN
  _eCheck                 := E_CHECK_STATE.AXIS_INFO_POINTER_INVALID;
  RETURN;
END_IF

IF NOT (_Data <> 0)
THEN
  _eCheck                 := E_CHECK_STATE.AXIS_DATA_POINTER_INVALID;
  RETURN;
END_IF

IF NOT (_NcParameterIn <> 0)
THEN
  _eCheck                 := E_CHECK_STATE.AXIS_NC_PARAMETER_POINTER_INVALID;
  RETURN;
END_IF

IF NOT (_NcParameterOut <> 0)
THEN
  _eCheck                 := E_CHECK_STATE.AXIS_NC_PARAMETER_POINTER_INVALID;
  RETURN;
END_IF

IF NOT (_HomeParameter <> 0)
THEN
  _eCheck                 := E_CHECK_STATE.AXIS_HOME_PARAMETER_POINTER_INVALID;
  RETURN;
END_IF

IF NOT (_GearInParameter <> 0)
THEN
  _eCheck                 := E_CHECK_STATE.AXIS_GEAR_IN_PARAMETER_POINTER_INVALID;
  RETURN;
END_IF
  
IF NOT (_MotionOptions <> 0)
THEN
  _eCheck                 := E_CHECK_STATE.AXIS_MOTION_OPTIONS_POINTER_INVALID;
  RETURN;
END_IF

IF NOT (_LimitSwitches <> 0)
THEN
  _eCheck                 := E_CHECK_STATE.AXIS_LIMIT_SWITCHES_POINTER_INVALID;
  RETURN;
END_IF

//-----------------------------------------------------------------------------
//  NaN INF check
//-----------------------------------------------------------------------------
IF NOT IsFinite(F_LReal(_Data^[_nAxisIndex].rSetPos))
THEN
	_Data^[_nAxisIndex].rSetPos     := 0.0;
END_IF

IF NOT IsFinite(F_LReal(_Data^[_nAxisIndex].rSetVelo))
THEN
	_Data^[_nAxisIndex].rSetVelo    := 0.0;
END_IF

IF NOT IsFinite(F_LReal(_Data^[_nAxisIndex].rAcc))
THEN
	_Data^[_nAxisIndex].rAcc        := 0.0;
END_IF

IF NOT IsFinite(F_LReal(_Data^[_nAxisIndex].rDec))
THEN
	_Data^[_nAxisIndex].rDec        := 0.0;
END_IF

IF NOT IsFinite(F_LReal(_Data^[_nAxisIndex].rOverride))
THEN
	_Data^[_nAxisIndex].rOverride   := 0.0;
END_IF
//-----------------------------------------------------------------------------
//-----------------------------------------------------------------------------
_eCheck                   := E_CHECK_STATE.CHECK_DONE;
Check                     := TRUE;
//-----------------------------------------------------------------------------
//-----------------------------------------------------------------------------
END_METHOD

//-------------------------------------------------------------------------------------
//
//  HAUD 2024 01 20
//
//  Cmd
//    - gets state for ctrl
//    - checks for eInit to be done, before any other commands are accepted
//    - prepare your commands here
//    - init what you have to here
//
//-------------------------------------------------------------------------------------
METHOD PRIVATE Cmd  : E_AXIS_STATE
VAR_INPUT
  eCmd              : E_AXIS_CTRL;
END_VAR
VAR_INST
  _estate   : E_AXIS_STATE;
  _stMsg    : ST_Message;
END_VAR

CASE eCmd
OF
  //-------------------------------------------------------------------------------------
  E_AXIS_CTRL.AXIS_INIT:
    _eInit    := _eResult             := AxisInit(FALSE);
    _estate                           := E_AXIS_STATE.AXIS_INIT;
ELSE
  IF (_eInit <> E_PROGRESS.PROGRESS_DONE)
  THEN
    _eResult                          := E_PROGRESS.PROGRESS_INIT;
    _estate                           := E_AXIS_STATE.AXIS_NO_INIT;
  ELSE
    CASE eCmd
    OF
      //---------------------------------------------------------------------------------
      E_AXIS_CTRL.AXIS_DISABLE:
        _eResult                      := AxisDisable(FALSE);
        _estate                       := E_AXIS_STATE.AXIS_DISABLE;

      //---------------------------------------------------------------------------------
      E_AXIS_CTRL.AXIS_ENABLE:
        _eResult                      := AxisEnable(FALSE);
        _estate                       := E_AXIS_STATE.AXIS_ENABLE;

      //---------------------------------------------------------------------------------
      E_AXIS_CTRL.AXIS_IDLE:
        _eResult                      := AxisBufferVelo(FALSE, _Data^[_nAxisIndex]);
        _eResult                      := AxisBufferPos(FALSE, _Data^[_nAxisIndex]);
        _eResult                      := AxisIdle(FALSE);
        _estate                       := E_AXIS_STATE.AXIS_IDLE;

      //---------------------------------------------------------------------------------
      E_AXIS_CTRL.AXIS_HOME:
        _eResult                      := AxisHome(FALSE);
        _estate                       := E_AXIS_STATE.AXIS_HOME;

      //---------------------------------------------------------------------------------
      E_AXIS_CTRL.AXIS_MOVE_POS:
        _eResult                      := AxisMoveToPosition(FALSE, _Data^[_nAxisIndex]);
        _estate                       := E_AXIS_STATE.AXIS_MOVE_POS;

      //---------------------------------------------------------------------------------
      E_AXIS_CTRL.AXIS_MOVE_VELO:
        _eResult                      := AxisMoveVelocity(FALSE, _Data^[_nAxisIndex]);
        _estate                       := E_AXIS_STATE.AXIS_MOVE_VELO;

      E_AXIS_CTRL.AXIS_SEND_TO_POS:
        _eResult                      := AxisSendToPosition(FALSE, _Data^[_nAxisIndex]);
        _estate                       := E_AXIS_STATE.AXIS_SEND_TO_POS;

      //---------------------------------------------------------------------------------
      E_AXIS_CTRL.AXIS_RESET:
        // OnChange clear error bit
        _Info^[_nAxisIndex].bError    := FALSE;
        _eResult                      := AxisReset(FALSE);
        _estate                       := E_AXIS_STATE.AXIS_RESET;

      //---------------------------------------------------------------------------------
      E_AXIS_CTRL.AXIS_HALT:
        _eResult                      := AxisHalt(FALSE, _Data^[_nAxisIndex]);
        _estate                       := E_AXIS_STATE.AXIS_HALT;

      //---------------------------------------------------------------------------------
      E_AXIS_CTRL.AXIS_STOP:
        _eResult                      := AxisStop(FALSE, _Data^[_nAxisIndex]);
        _estate                       := E_AXIS_STATE.AXIS_STOP;


      //---------------------------------------------------------------------------------
      E_AXIS_CTRL.AXIS_MOVE_BUFFER:
        _eResult                      := AxisBufferPos(FALSE, _Data^[_nAxisIndex]);
        _estate                       := E_AXIS_STATE.AXIS_MOVE_BUFFER;


      //---------------------------------------------------------------------------------
      E_AXIS_CTRL.AXIS_MOVE_BUFFER_VELO:
        _eResult                      := AxisBufferVelo(FALSE, _Data^[_nAxisIndex]);
        _estate                       := E_AXIS_STATE.AXIS_MOVE_BUFFER_VELO;


      //---------------------------------------------------------------------------------
      E_AXIS_CTRL.AXIS_PARAMETER_READ:
        _eParameterNrRead             := _NcParameterIn^[_nAxisIndex].ParameterNumber;

        _eResult                      := AxisParameterRead(FALSE, _eParameterNrRead);
        _estate                       := E_AXIS_STATE.AXIS_PARAMETER_READ;


      //---------------------------------------------------------------------------------
      E_AXIS_CTRL.AXIS_PARAMETER_WRITE:
        _eParameterNrWrite            := _NcParameterIn^[_nAxisIndex].ParameterNumber;
        _rParameterWrtValue           := _NcParameterIn^[_nAxisIndex].rValue;
        _eResult                      := AxisParameterWrite(FALSE, _eParameterNrWrite);
        _estate                       := E_AXIS_STATE.AXIS_PARAMETER_WRITE;


      //---------------------------------------------------------------------------------
      E_AXIS_CTRL.AXIS_PARAMETER_WRITE_PERSISTENT:
        _eParameterNrWrite            := _NcParameterIn^[_nAxisIndex].ParameterNumber;
        _rParameterWrtValue           := _NcParameterIn^[_nAxisIndex].rValue;
        _eResult                      := AxisParameterWritePersistent(FALSE, _eParameterNrWrite);
        _estate                       := E_AXIS_STATE.AXIS_PARAMETER_WRITE_PERSISTENT;

      //---------------------------------------------------------------------------------
      E_AXIS_CTRL.AXIS_GEAR_IN:
        _eResult                      := AxisGearIn(FALSE);
        _estate                       := E_AXIS_STATE.AXIS_GEAR_IN;

      //---------------------------------------------------------------------------------    
      E_AXIS_CTRL.AXIS_GEAR_OUT:
        _eResult                      := AxisGearOut(FALSE);
        _estate                       := E_AXIS_STATE.AXIS_GEAR_OUT;

      //---------------------------------------------------------------------------------
      E_AXIS_CTRL.AXIS_GEAR_IN_MULTIMASTER:
        _fbGearInMultiMaster.Master1  := _MultiMasterDummyRef[1];
        _fbGearInMultiMaster.Master2  := _MultiMasterDummyRef[2];
        _fbGearInMultiMaster.Master3  := _MultiMasterDummyRef[3];
        _fbGearInMultiMaster.Master4  := _MultiMasterDummyRef[4];

        _eResult                      := AxisGearInMultiMaster(FALSE);
        _estate                       := E_AXIS_STATE.AXIS_GEAR_IN_MULTIMASTER;

    //-----------------------------------------------------------------------------------
    ELSE
      _estate                         := E_AXIS_STATE.AXIS_NULL;

      IF (eCmd = E_AXIS_CTRL.AXIS_NULL)
      THEN
        _eResult                      := E_PROGRESS.PROGRESS_DONE;
      ELSE
        _eResult                      := E_PROGRESS.PROGRESS_INVALID;
  
        _stMsg.eType                  := E_MessageType.eMessageError;
        _stMsg.eDevice                := E_Device.Axis + (_Axes[_nAxisIndex].NcToPlc.AxisId);
        _stMsg.eSubdevice             := e_Subdevice.AxisControl;
        _stMsg.iErrorNumber           := 0;
  
        _stMsg.sText                  := 'E_AXIS_CTRL.';
        _stMsg.sText                  := concat(_stMsg.sText, TO_STRING(eCmd));
        _stMsg.sText                  := concat(_stMsg.sText, ': ');
        _stMsg.sText                  := concat(_stMsg.sText, TO_STRING(_eResult));

        f_MessageSet(_stMsg);
      END_IF
    END_CASE
  END_IF // _eInit
END_CASE

Cmd                                   := _estate;
END_METHOD

METHOD PRIVATE GetCalibrationCam : BOOL
VAR_INST
  _bCal     : Bool;
END_VAR
IF NOT Check() THEN RETURN; END_IF

IF _HomeParameter^[_nAxisIndex].stHomingParam.SimulateHomeSensor
THEN
	IF (_AxisRef.NcToPlc.HomingState < 4)
  THEN
		_bCal := TRUE;
	ELSE
		_bCal := FALSE;
	END_IF
ELSIF _HomeParameter^[_nAxisIndex].stHomingParam.HomeOnLimitMin
THEN
	_bCal := _LimitSwitches^[_nAxisIndex].bMinimum   XOR 
           _HomeParameter^[_nAxisIndex].stHomingParam.InvertHomeSensor;

ELSIF _HomeParameter^[_nAxisIndex].stHomingParam.HomeOnLimitMax
THEN
	_bCal := _LimitSwitches^[_nAxisIndex].bMaximum   XOR 
           _HomeParameter^[_nAxisIndex].stHomingParam.InvertHomeSensor;
ELSE
	_bCal := _LimitSwitches^[_nAxisIndex].bCalibrate XOR 
           _HomeParameter^[_nAxisIndex].stHomingParam.InvertHomeSensor;
END_IF

GetCalibrationCam := _bCal;
END_METHOD

PROPERTY HomingParameter : pointer to ARRAY[1..PLC_CONSTANT.MAX_AXIS] OF st_homing
SET
_HomeParameter := HomingParameter;
END_SET
END_PROPERTY

PROPERTY LimitSwitches : pointer to ARRAY[1..PLC_CONSTANT.MAX_AXIS] OF ST_AXIS_LIMIT_SWITCHES
SET
_LimitSwitches := LimitSwitches;
END_SET
END_PROPERTY

METHOD PRIVATE LogControl
VAR_INST
  _sResult,
  _sCtrl            : STRING(60);

  _stMsg            : ST_Message;
END_VAR
  _stMsg.eType               := E_MessageType.eMessageInfo;
  _stMsg.eDevice             := E_Device.Axis + (_AxisRef.NcToPlc.AxisId);
  _stMsg.eSubdevice          := e_Subdevice.AxisControl;
  _stMsg.iErrorNumber        := _nAxisIndex;

  _sCtrl                     := concat('E_AXIS_CTRL', '.');
  _sCtrl                     := concat(_sCtrl, TO_STRING(_eCmd));

  _stMsg.sText               := concat('new command: ', _sCtrl);

  IF (_MessageLevel > E_MessageType.eMessageError)
  THEN
    f_MessageSet(_stMsg);
  END_IF
END_METHOD

METHOD PRIVATE LogResult
VAR_INST
  _sResult,
  _sCtrl            : STRING(60);

  _stMsg            : ST_Message;
END_VAR

  _stMsg.eType               := E_MessageType.eMessageInfo;
  _stMsg.eDevice             := E_Device.Axis + (_AxisRef.NcToPlc.AxisId);
  _stMsg.eSubdevice          := e_Subdevice.AxisControl;
  _stMsg.iErrorNumber        := _nAxisIndex;

  _sCtrl                     := concat('E_AXIS_CTRL', '.');
  _sCtrl                     := concat(_sCtrl, TO_STRING(_eCmd));

  _sResult                   := TO_STRING(_eResult);

  _stMsg.sText               := concat(_sCtrl, ': ');
  _stMsg.sText               := concat(_stMsg.sText, _sResult);

  IF (_MessageLevel > E_MessageType.eMessageError)
  THEN
    f_MessageSet(_stMsg);
  END_IF
END_METHOD

PROPERTY MotionOptions : pointer to ARRAY[1..PLC_CONSTANT.MAX_AXIS] OF ST_MOTION_OPTIONS
SET
_MotionOptions := MotionOptions;
END_SET
END_PROPERTY

PROPERTY NcParameterIn : pointer to ARRAY[1..PLC_CONSTANT.MAX_AXIS] OF st_nc_parameter
SET
_NcParameterIn := NcParameterIn;
END_SET
END_PROPERTY

PROPERTY NcParameterOut : pointer to ARRAY[1..PLC_CONSTANT.MAX_AXIS] OF st_nc_parameter
SET
_NcParameterOut := NcParameterOut;
END_SET
END_PROPERTY

PROPERTY NcParameterValue : Lreal
GET
NcParameterValue := _rParameterReadValue;
END_GET
END_PROPERTY

METHOD PRIVATE ResetSoE : E_PROGRESS
VAR_INPUT
  Execute           : BOOL;
END_VAR
VAR_INST
  _eState           : E_PROGRESS;
  _rValue           : LREAL;
  _udiErrSer,
  _udiErrAds        : UDINT;
  _stMsg            : ST_Message;

	_fbReset		      : Tc2_MC2_Drive.FB_SoEReset;
  _tonDelay         : Tc2_Standard.TON;
	_nRepeat			    : UINT;

  _sErrorSercos     : Tc2_System.T_MaxString;

END_VAR
IF NOT Check() THEN ResetSoE := E_PROGRESS.PROGRESS_ERROR; RETURN; END_IF
IF NOT Execute THEN _eState := E_PROGRESS.PROGRESS_INIT; END_IF

CASE _eState
OF
  E_PROGRESS.PROGRESS_INIT:
    IF Execute 
    THEN
      memset(ADR(_stMsg),0,SIZEOF(_stMsg));
      memset(ADR(_sErrorSercos),0,SIZEOF(_sErrorSercos));

		  _nRepeat                      := 1;
      _udiErrSer := _udiErrAds      := 0;
      _rValue                       := 0;
      _eState                       := E_PROGRESS.PROGRESS_BUSY;
    END_IF
END_CASE
CASE _eState
OF
  E_PROGRESS.PROGRESS_BUSY:
    _eState                         := E_PROGRESS.PROGRESS_OCCUPIED;
		_tonDelay(
            IN                      := FALSE);

		_fbReset(
            Execute                 := FALSE, 
            Timeout                 := T#2500MS, 
            Axis                    := _AxisRef);
END_CASE
CASE _eState
OF
  E_PROGRESS.PROGRESS_OCCUPIED:
		_tonDelay(
            PT                      := T#1500MS, 
            IN                      := TRUE);

		_fbReset(
            Execute                 := TRUE, 
            Axis                    := _AxisRef, 
            AdsErrId                => _udiErrAds, 
            SercosErrId             => _udiErrSer);

    IF _fbReset.Error
    THEN
      _stMsg.eType                  := E_MessageType.eMessageError;
      _stMsg.eDevice                := e_Device.Axis + (_AxisRef.NcToPlc.AxisId);
      _stMsg.eSubdevice             :=  e_SubDevice.fbResetSercos;
      _stMsg.iErrorNumber           := _udiErrAds;

      _sErrorSercos                 := Tc2_Utilities.DATA_TO_HEXSTR(ADR(_udiErrSer), SIZEOF(_udiErrSer), FALSE);

      _stMsg.sText                  := concat('Sercos Err Nr: ', _sErrorSercos);

      f_MessageSet(_stMsg);

      _Info^[_nAxisIndex].nErrorId := _udiErrSer;
      _eState                       := E_PROGRESS.PROGRESS_ERROR;

		ELSIF NOT _fbReset.Busy
		THEN
      _eState                       := E_PROGRESS.PROGRESS_WORKING;

    ELSE
      IF _tonDelay.Q AND
         _AxisRef.NcToPlc.StateDWord.28
      THEN
        _nRepeat                    := _nRepeat + 1;
        _eState                     := E_PROGRESS.PROGRESS_BUSY;    
      END_IF

      IF (_nRepeat > 5)
      THEN
        _eState                     := E_PROGRESS.PROGRESS_ERROR;
      END_IF
		END_IF
END_CASE
CASE _eState
OF
  E_PROGRESS.PROGRESS_WORKING:
    _eState                         := E_PROGRESS.PROGRESS_DONE;
END_CASE


ResetSoE := _eState;
END_METHOD

PROPERTY TargetWindow : lreal
GET
END_GET
SET
END_SET
END_PROPERTY

END_FUNCTION_BLOCK

// ---- _MSG/class/fb_MessageData.TcPOU
FUNCTION_BLOCK ABSTRACT fb_MessageData IMPLEMENTS I_MessageData
VAR CONSTANT
{attribute 'hide'}
  STR_LEN       : UDINT := 524_288;
END_VAR
VAR
  _eCheck       : E_MESSAGE_CHECK;            // pointer check state

  _pFileRoot    : POINTER TO STRING(255);     // you decide (example in GVL_MSG.LOG_FILE)
  _pDirRoot     : POINTER TO STRING(255);     // see GVL_MSG.LOG_DIR

  _nMsgIndex    : REFERENCE TO UINT;          // Hypnos IS the only one in the village, if there are more you need more villages
  _nErrIndex    : REFERENCE TO UINT;          // Thanatos, Hypnos stern and more serious brother

  _dtLocalTime  : POINTER TO DT;
  _pMsgList     : POINTER TO ARRAY[1..GVL_MSG_AXIS.MAX_MESSAGE] OF ST_Message; // attach your list here

	_rtrigReset   : Tc2_Standard.R_TRIG;
	_aWriteList   : ARRAY[1..GVL_MSG_AXIS.MAX_MESSAGE] OF ST_Message;
	_sWriteData   : STRING(STR_LEN);
	_sNewLine     : STRING := '$N';
	_sTab         : STRING := '$T';
	_iCount, 
	_iStart, 
	_iEnd         : UINT;

	_fbCreateDir  : Tc2_System.FB_CreateDir;
	_sTmp         : STRING(256);
	_sFilename    : STRING(256);
	_sFolderDate  : STRING;
	_bFileCreated : BOOL;

	_fbFileOpen   : Tc2_System.FB_FileOpen;
	_fbFileWrite  : Tc2_System.FB_FileWrite;
	_fbFileClose  : Tc2_System.FB_FileClose;
END_VAR

METHOD Builder : BOOL // string concat for length > 255
VAR_INPUT
  pInString   : POINTER TO STRING;
  pOutString  : POINTER TO STRING(STR_LEN);
  Length      : UINT;
END_VAR
VAR
  Counter     : UDINT;
  pInWork     : POINTER TO BYTE;
  pOutWork    : POINTER TO BYTE;
END_VAR
pOutWork := pOutString;
pInWork := pInString;
Counter := 0;

(*check termination*)
WHILE (pOutWork^ <> 0) AND
      (Counter < STR_LEN+1)
DO
  Counter := Counter + 1;
  pOutWork := pOutWork + 1;
END_WHILE

(* append only if data fits into output *)
IF (Counter + Length < STR_LEN+1)
THEN

  (* append data *)
  FOR Counter := 1 TO Length
  DO
    pOutWork^ := pInWork^;
    pOutWork := pOutWork + 1;
    pInWork := pInWork + 1;
  END_FOR

  (* terminate *)
  pOutWork := pOutWork + 1;
  pOutWork^ := 0;
END_IF
END_METHOD

METHOD Check : BOOL
VAR_INPUT
END_VAR

IF NOT (_dtLocalTime <> 0)
THEN
  _eCheck       := E_MESSAGE_CHECK.MSG_CHECK_INVALID_POINTER_TIME;
  RETURN;
END_IF

IF NOT (_pMsgList <> 0)
THEN
  _eCheck       := E_MESSAGE_CHECK.MSG_CHECK_INVALID_POINTER_LIST;
  RETURN;
END_IF

IF NOT (_pFileRoot <> 0)
THEN
  _eCheck       := E_MESSAGE_CHECK.MSG_CHECK_INVALID_POINTER_ROOT_FILE;
  RETURN;
END_IF

IF NOT (_pDirRoot <> 0)
THEN
  _eCheck       := E_MESSAGE_CHECK.MSG_CHECK_INVALID_POINTER_ROOT_DIR;
  RETURN;
END_IF

IF NOT __ISVALIDREF(_nMsgIndex)
THEN
  _eCheck       := E_MESSAGE_CHECK.MSG_CHECK_INVALID_POINTER_MSG_IDX;
  RETURN;
END_IF

IF NOT __ISVALIDREF(_nErrIndex)
THEN
  _eCheck       := E_MESSAGE_CHECK.MSG_CHECK_INVALID_POINTER_ERR_IDX;
  RETURN;
END_IF


_eCheck         := E_MESSAGE_CHECK.MSG_CHECK_DONE;
Check           := TRUE;
END_METHOD

METHOD Device_to_String : string
VAR_INPUT
  eMsgDevice    : e_Device;
END_VAR
VAR
  sId                 : STRING := '_ID_';
  nId                 : UDINT;
END_VAR
IF (eMsgDevice < e_device.General)
THEN
  // below general case
  nId := TO_UDINT(eMsgDevice);
  sId := concat(sId, TO_STRING(nId));

  Device_to_String := TO_STRING(eMsgDevice);

ELSE
  IF (eMsgDevice >= e_Device.DataProduct)
  THEN
    nId := eMsgDevice MOD e_Device.DataProduct;
    sId := concat(sId, TO_STRING(nId));
 
    Device_to_String := concat(TO_STRING(e_Device.DataProduct), sId);

  ELSIF (eMsgDevice >= e_Device.Application)
  THEN
    nId := eMsgDevice MOD e_Device.Application;
    sId := concat(sId, TO_STRING(nId));
 
    Device_to_String := concat(TO_STRING(e_Device.Application), sId);

  ELSIF (eMsgDevice >= e_Device.TicketListCtrl)
  THEN
    nId := eMsgDevice MOD e_Device.TicketListCtrl;
    sId := concat(sId, TO_STRING(nId));
 
    Device_to_String := concat(TO_STRING(e_Device.TicketListCtrl), sId);

  ELSIF (eMsgDevice >= e_Device.ProcessListCtrl)
  THEN
    nId := eMsgDevice MOD e_Device.ProcessListCtrl;
    sId := concat(sId, TO_STRING(nId));
 
    Device_to_String := concat(TO_STRING(e_Device.ProcessListCtrl), sId);

  ELSIF (eMsgDevice >= e_Device.Process)
  THEN
    nId := eMsgDevice MOD e_Device.Process;
    sId := concat(sId, TO_STRING(nId));
 
    Device_to_String := concat(TO_STRING(e_Device.Process), sId);

  ELSIF (eMsgDevice >= e_Device.FlyingSaw)
  THEN
    nId := eMsgDevice MOD e_Device.FlyingSaw;
    sId := concat(sId, TO_STRING(nId));
 
    Device_to_String := concat(TO_STRING(e_device.FlyingSaw), sId);

  ELSIF (eMsgDevice >= e_Device.MetricsAxis)
  THEN
    nId := eMsgDevice MOD e_Device.MetricsAxis;
    sId := concat(sId, TO_STRING(nId));
 
    Device_to_String := concat(TO_STRING(e_device.MetricsAxis), sId);

  ELSIF (eMsgDevice >= e_Device.MetricsXts)
  THEN
    nId := eMsgDevice MOD e_Device.MetricsXts;
    sId := concat(sId, TO_STRING(nId));
 
    Device_to_String := concat(TO_STRING(e_device.MetricsXts), sId);

  ELSIF (eMsgDevice >= e_device.XfcAxis)
  THEN
    nId := eMsgDevice MOD e_device.XfcAxis;
    sId := concat(sId, TO_STRING(nId));
 
    Device_to_String := concat(TO_STRING(e_device.XfcAxis), sId);

  ELSIF (eMsgDevice >= e_device.Axis)
  THEN
    nId := eMsgDevice MOD e_device.Axis;
    sId := concat(sId, TO_STRING(nId));
 
    Device_to_String := concat(TO_STRING(e_device.Axis), sId);

  ELSIF (eMsgDevice >= e_device.NciChannelCtrl)
  THEN
    nId := eMsgDevice MOD e_device.NciChannelCtrl;
    sId := concat(sId, TO_STRING(nId));
 
    Device_to_String := concat(TO_STRING(e_device.NciChannelCtrl), sId);

  ELSIF (eMsgDevice >= e_device.NciChannel)
  THEN
    nId := eMsgDevice MOD e_device.NciChannel;
    sId := concat(sId, TO_STRING(nId));
 
    Device_to_String := concat(TO_STRING(e_device.NciChannel), sId);

  ELSIF (eMsgDevice >= e_Device.Camming)
  THEN
    nId := eMsgDevice MOD e_Device.Camming;
    sId := concat(sId, TO_STRING(nId));
 
    Device_to_String := concat(TO_STRING(e_device.Camming), sId);

  ELSIF (eMsgDevice >= e_Device.XtsStation)
  THEN
    nId := eMsgDevice MOD e_Device.XtsStation;
    sId := concat(sId, TO_STRING(nId));
 
    Device_to_String := concat(TO_STRING(e_device.XtsStation), sId);

  ELSIF (eMsgDevice >= e_Device.XfcTouchProbe)
  THEN
    nId := eMsgDevice MOD e_Device.XfcTouchProbe;
    sId := concat(sId, TO_STRING(nId));
 
    Device_to_String := concat(TO_STRING(e_device.XfcTouchProbe), sId);

  ELSIF (eMsgDevice >= e_Device.XfcTriggerBox)
  THEN
    nId := eMsgDevice MOD e_Device.XfcTriggerBox;
    sId := concat(sId, TO_STRING(nId));
 
    Device_to_String := concat(TO_STRING(e_device.XfcTriggerBox), sId);

  ELSIF (eMsgDevice >= e_Device.XtsTransportUnit)
  THEN
    nId := eMsgDevice MOD e_Device.XtsTransportUnit;
    sId := concat(sId, TO_STRING(nId));
 
    Device_to_String := concat(TO_STRING(e_device.XtsTransportUnit), sId);

  ELSIF (eMsgDevice >= e_Device.MoverCtrl)
  THEN
    nId := eMsgDevice MOD e_Device.MoverCtrl;
    sId := concat(sId, TO_STRING(nId));
 
    Device_to_String := concat(TO_STRING(e_device.MoverCtrl), sId);

  ELSIF (eMsgDevice >= e_Device.Mover)
  THEN
    nId := eMsgDevice MOD e_Device.Mover;
    sId := concat(sId, TO_STRING(nId));
 
    Device_to_String := concat(TO_STRING(e_device.Mover), sId);

  ELSIF (eMsgDevice >= e_Device.XpuCtrl)
  THEN
    nId := eMsgDevice MOD e_Device.XpuCtrl;
    sId := concat(sId, TO_STRING(nId));
 
    Device_to_String := concat(TO_STRING(e_device.XpuCtrl), sId);

  ELSIF (eMsgDevice >= e_Device.Xpu)
  THEN
    nId := eMsgDevice MOD e_Device.Xpu;
    sId := concat(sId, TO_STRING(nId));
 
    Device_to_String := concat(TO_STRING(e_device.Xpu), sId);

  ELSIF (eMsgDevice >= e_Device.CaGroup)
  THEN
    nId := eMsgDevice MOD e_Device.CaGroup;
    sId := concat(sId, TO_STRING(nId));
 
    Device_to_String := concat(TO_STRING(e_device.CaGroup), sId);

  ELSIF (eMsgDevice >= e_Device.General)
  THEN
    nId := eMsgDevice MOD e_Device.General;
    sId := concat(sId, TO_STRING(nId));
 
    Device_to_String := concat(TO_STRING(e_device.General), sId);

  ELSE
    Device_to_String := TO_STRING(eMsgDevice);
  END_IF
END_IF
END_METHOD

PROPERTY DirRoot : POINTER to string(255)
SET
_pDirRoot := DirRoot;
END_SET
END_PROPERTY

PROPERTY ErrorIndex : reference to uint
SET
_nErrIndex  REF= ErrorIndex;
END_SET
END_PROPERTY

PROPERTY FileRoot : pointer to string(255)
SET
_pFileRoot := FileRoot;
END_SET
END_PROPERTY

METHOD FolderDate : STRING
VAR_INPUT
	LocalTime   : POINTER TO DT;
END_VAR
VAR
	sTmp        : STRING;
END_VAR
IF NOT (LocalTime <> 0)
THEN
	FolderDate := 'NULL';
	RETURN;
END_IF

sTmp := DT_TO_STRING(LocalTime^);

// cut off #dt literal
sTmp := right(sTmp, len(sTmp)-3);

sTmp := replace(sTmp, '_', 1, 5);
sTmp := replace(sTmp, '_', 1, 8);

sTmp := left(sTmp,10);	// year_month_day

FolderDate := sTmp;
END_METHOD

PROPERTY LocalTime : pointer to DT
SET
_dtLocalTime := LocalTime;
END_SET
END_PROPERTY

PROPERTY MessageIndex : reference to uint
SET
_nMsgIndex   REF= MessageIndex;
END_SET
END_PROPERTY

PROPERTY MsgList : pointer to ARRAY[1..GVL_MSG_AXIS.MAX_MESSAGE] OF st_message
SET
_pMsgList := MsgList;
END_SET
END_PROPERTY

METHOD StringLen : UINT // 	string length for len > 255
VAR_INPUT
  pInString		: POINTER TO STRING(STR_LEN);
END_VAR
VAR
	Counter			: UINT;
	pInWork			: POINTER TO BYTE;
END_VAR
pInWork := pInString;
Counter := 0;

WHILE (pInWork^ <> 0) AND
			(Counter < STR_LEN)
DO
	Counter := Counter + 1;
	pInWork := pInWork + 1;
END_WHILE

StringLen := Counter;
END_METHOD

METHOD WriteData  : e_progress
VAR_INPUT
  bExecute        : BOOL;
END_VAR
VAR_INST
  _eState         : e_progress;
  _bError         : BOOL;
  _nErrorId       : UDINT;
END_VAR
IF NOT bExecute
THEN
  _eState                     := E_PROGRESS.PROGRESS_INIT;
END_IF

CASE _eState 
OF

	E_PROGRESS.PROGRESS_INIT:
		_fbFileOpen.bExecute      := FALSE;
		_fbFileWrite.bExecute	    := FALSE;
		_fbFileClose.bExecute	    := FALSE;

		IF bExecute
		THEN
      _nErrorId               := 0;
      _eState                 := E_PROGRESS.PROGRESS_BUSY;
		END_IF

	E_PROGRESS.PROGRESS_BUSY:
		_fbFileOpen.bExecute      := TRUE;

    IF _fbFileOpen.bError
    THEN
		  _fbFileOpen.bExecute    := FALSE;
      _nErrorId               := _fbFileOpen.nErrId;
      _eState                 := E_PROGRESS.PROGRESS_ERROR;

		ELSIF _fbFileOpen.bBusy
		THEN
      _eState                 := E_PROGRESS.PROGRESS_PREPARE;
		END_IF

	E_PROGRESS.PROGRESS_PREPARE:
		IF NOT _fbFileOpen.bBusy
		THEN
		  _fbFileOpen.bExecute    := FALSE;
			_fbFileWrite.bExecute   := TRUE;
      _eState                 := E_PROGRESS.PROGRESS_STARTUP;
		END_IF

	E_PROGRESS.PROGRESS_STARTUP:
    IF _fbFileWrite.bError
    THEN
			_fbFileWrite.bExecute   := FALSE;
      _nErrorId               := _fbFileWrite.nErrId;
      _eState                 := E_PROGRESS.PROGRESS_ERROR;

		ELSIF _fbFileWrite.bBusy
		THEN
      _eState                 := E_PROGRESS.PROGRESS_CHECK;
		END_IF

	E_PROGRESS.PROGRESS_CHECK:
		IF NOT _fbFileWrite.bBusy
		THEN
			_fbFileWrite.bExecute   := FALSE;
			_fbFileClose.bExecute   := TRUE;
      _eState                 := E_PROGRESS.PROGRESS_OCCUPIED;
		END_IF

	E_PROGRESS.PROGRESS_OCCUPIED:
    IF _fbFileClose.bError
    THEN
			_fbFileClose.bExecute   := FALSE;
      _nErrorId               := _fbFileClose.nErrId;
      _eState                 := E_PROGRESS.PROGRESS_ERROR;

		ELSIF _fbFileClose.bBusy
		THEN
      _eState                 := E_PROGRESS.PROGRESS_WORKING;
		END_IF

	E_PROGRESS.PROGRESS_WORKING:
		IF NOT _fbFileClose.bBusy
		THEN
			_fbFileClose.bExecute   := FALSE;
      _eState                 := E_PROGRESS.PROGRESS_DONE;
		END_IF
END_CASE


_fbFileOpen(
	sNetId:= , 
	sPathName:= _sFilename, 
	nMode:= FOPEN_MODEAPPEND OR FOPEN_MODEPLUS, 
	ePath:= PATH_GENERIC, 
	bExecute:= , 
	tTimeout:= T#10S, 
	bBusy=> , 
	bError=> , 
	nErrId=> , 
	hFile=> );

_fbFileWrite(
	sNetId:= , 
	hFile:= _fbFileOpen.hFile, 
	pWriteBuff:= ADR(_sWriteData), 
	cbWriteLen:= StringLen(ADR(_sWriteData)), 
	bExecute:= , 
	tTimeout:= T#10S, 
	bBusy=> , 
	bError=> , 
	nErrId=> , 
	cbWrite=> );

_fbFileClose(
	sNetId:= , 
	hFile:= _fbFileOpen.hFile, 
	bExecute:= , 
	tTimeout:= T#10S, 
	bBusy=> , 
	bError=> , 
	nErrId=> );

WriteData                     := _eState;
END_METHOD

END_FUNCTION_BLOCK

// ---- PLC_MOTION/_GVL/GlobalTextList.TcGTLO
TEXTLIST GlobalTextList
  526 = 'Activate'
  315 = 'eDevice'
  316 = 'eSubdevice'
  314 = 'eType'
  317 = 'iErrorNumber'
  319 = 'sText'
  318 = 'tTime'
  517 = 'WRITE TO FILE'
END_TEXTLIST

// ---- _MSG/types/TL_E_MESSAGETYPE.TcTLO
TEXTLIST TL_E_MESSAGETYPE
  0 = 'eMessageEmpty'
  1 = 'eMessageError'
  2 = 'eMessageWarning'
  3 = 'eMessageInfo'
  4 = 'eMessageVerbose'
   = ''
END_TEXTLIST
